// TIA Portal V17 export
// export: Created 2025-03-05T08:00:31.4728313Z, ExportSetting WithDefaults, DisplayName Totally Integrated Automation Portal, DisplayVersion V17 Update 8, DisplayName TIA Portal Openness, DisplayVersion V17 Update 8, DisplayName TIA Portal Version Control Interface, DisplayVersion V17, DisplayName SINAMICS Startdrive Advanced, DisplayVersion V17 SP2, DisplayName SINAMICS Startdrive G110M, G120, G120C, G120D, G120P, G115D, DisplayVersion V17 SP2, DisplayName SINAMICS Startdrive G130, G150, S120, S150, SINAMICS MV, S210, DisplayVersion V17 SP2, DisplayName STEP 7 Professional, DisplayVersion V17 Update 8, DisplayName SINUMERIK ONE STEP 7 Toolbox, DisplayVersion V17 Update 12, DisplayName SINUMERIK 840D sl STEP 7 Toolbox, DisplayVersion V17 Update 12, DisplayName STEP 7 Safety, DisplayVersion V17 Update 6, DisplayName WinCC Advanced, DisplayVersion V17 Update 8
DATA_BLOCK "DB1223_MAINTENANCE_UNIT_01_CLADDING"   // DB1223
{ S7_Optimized_Access := 'FALSE'; DB_Accessible_From_OPC_UA := 'FALSE' }
AUTHOR : ETXETAR
VERSION : 1.0
// stored: AutoNumber false, DBAccessibleFromOPCUA false, DBAccessibleFromWebserver true, IsOnlyStoredInLoadMemory false, IsWriteProtectedInAS false
   VAR RETAIN
      SEQUENCE : "RUN_CNC_SEQ";
      TIMER_RESET_AUX_HEAD_COVER { S7_SetPoint := 'True'} : TON_TIME;   // TIMER RESET AUX HEAD PROTECTION COVER
      "REQUEST PULSE COUNTER" : CTU_INT;   // REQUEST PULSE COUNTER
   END_VAR
BEGIN
   SEQUENCE.TIMER_TIME_EXCEED.PT := T#180s;
   TIMER_RESET_AUX_HEAD_COVER.PT := T#30S;
END_DATA_BLOCK
